FUNCTION_BLOCK FB_RotateStation IMPLEMENTS I_StationProcess
VAR
	_StationAngle  : LREAL;
	_NumberOfTurns : DINT;

END_VAR

METHOD Execute : BOOL
VAR_INPUT
	Mover	: XPlanarApplication.I_XPlanarMover;
END_VAR

VAR_INST
	CommandResult : I_PlanarTaskResult;
END_VAR
CommandResult := Mover.MoveCommand.Rotate(_StationAngle, _NumberOfTurns);
IF CommandResult.Done THEN
	Execute := TRUE;
ELSIF CommandResult.Error THEN
	; //Command returned an error, DO SOMETHING!
END_IF
END_METHOD

PROPERTY NumberOfTurns : DINT
SET
_NumberOfTurns := NumberOfTurns;
END_SET
END_PROPERTY

PROPERTY StationAngle : LREAL
SET
_StationAngle := StationAngle;
END_SET
END_PROPERTY

END_FUNCTION_BLOCK

(* stored: Version 1.1.0.1
   POU FB_RotateStation: Id {d0ee9b9c-eeff-4082-9db1-0bc32eab28c5}, SpecialFunc None
   Method Execute: Id {37584313-51fc-4c4e-9c14-700cf13d2d8a}
   Property NumberOfTurns: Id {9d661a2e-f7f3-4558-afb3-350c215cc0c4}
   Set Set: Id {cad60f88-e9df-4e9a-94e5-e7e43cc8e24a}
   Property StationAngle: Id {568cd894-6b94-4015-b665-4e2c3332f5de}
   Set Set: Id {8b016c78-79fe-4d2f-b17c-5ed06ac7ec95} *)
